{attribute 'GeneratedUsingTerminal: EP7041-0002-0016'}
{attribute addProperty BoxType "EP7041-0002-0016"}
{attribute addProperty Id "StatusAT %I*Status_B679584511"}
{attribute addProperty CRC "921504111"}
{attribute addProperty Size "11"}
TYPE STM_Status_36ED096F :
STRUCT
	{attribute addProperty Name "Status"}
	Status AT %I* : Status_B6795845;
END_STRUCT
END_TYPE

(* stored: Version 1.2.0.0, ProductVersion 3.1.4024.9
   DUT STM_Status_36ED096F: Id {1c9980aa-bb8d-4921-8640-9a830fb87530} *)
